// TIA Portal V20 export
VAR_GLOBAL   // PLC tag table "LGR_Const_RobotNumber"
END_VAR
VAR_GLOBAL CONSTANT   // user constants
   GR1 : USInt := 1;
   GR2 : USInt := 2;
   GR3 : USInt := 3;
   All_GR : USInt := 10;
END_VAR
